PROGRAM MAIN
VAR
	Timer1 :TON;
	Timer2 : TON;
	Timer3 : TON;
	PulseTimer1 : TP;

	CurrentState  : States;
	
	ServoRTrigY : R_Trig ; 
	ServoRTrigX : R_Trig ; 
	
	//Eigen trigger booleans
	InitYReady : BOOL;
	InitXReady : BOOL;
	droppingDown : BOOL; //test
	
	TimerTest1 : TIME;
	TimerResult : TIME;
	
	Move_Arm : MoveArm;
	Count_Free_Spaces : CountFreeSpaces;
	Find_Free : FindFree;
	
	PalletArray: ARRAY [1..25] OF BOOL := [25(FALSE)];
	Pos : INT;
	
	DrinkArray: ARRAY [1..25] OF Drinks := [25(Drinks.Cola)]; 
	FreeCola : INT;
	FreeFanta : INT;
	
	//messages voor Nicky & Jens
	BottleAvailable : BOOL;
	NoCover : BOOL;
	NoBottle : BOOL;
	ColaFanta: INT;
	

	
END_VAR

PulseTimer1(IN:=GVL_IO.Start_button, PT:=T#150MS);
Timer1(IN:= GVL_IO.a_1_Vertical_Zaxis_downward, PT:= T#10MS);
Timer2(IN:=GVL_IO.a_1_Vertical_Zaxis_downward, PT:=T#10MS);
Timer3(IN:=droppingDown AND NOT GVL_IO.a_1_Vertical_Zaxis_downward, PT:=T#280MS);

CASE CurrentState OF
States.Init:
		//Aanzetten van servo's. Dit kan even duren GEEN HOMING
		GVL_IO.SVONX_SERVO_ON_tableX 	  := TRUE; 
		GVL_IO.SVONY_SERVO_ON_translY 	  := TRUE;
		
		GVL_IO.SETUPX_ORIGIN_tableX := PulseTimer1.Q;
		GVL_IO.SETUPY_ORIGIN_translY := PulseTimer1.Q;
		
		//// Koppelen van outputs Busy aan var's. Triggered op een falling edge.
		IF PulseTimer1.Q THEN
			ServoRTrigX ( clk := gvl_io.SETONX_ORIGIN_tableX ); 
	  		ServoRTrigY ( clk := gvl_io.SETONY_ORIGIN_translationY );
		END_IF
		
		// Bools setten aan de hand van triggers.
		IF ServoRTrigX.Q THEN
			InitXReady:= TRUE;
		END_IF
		
		IF ServoRTrigY.Q THEN
			InitYReady:= TRUE;
		END_IF
		
		// Init voltooid ga naar idle
		IF InitXReady AND InitYReady THEN
			Pos:= 1;
			NoCover := FALSE;
			NoBottle := FALSE;
			ColaFanta := drinks.Cola;
			CurrentState:= States.Idle;
		END_IF
		
States.Idle:
		//TEST =========================================================
		IF NOT GVL_IO.Stop_button THEN
			BottleAvailable := TRUE;
		END_IF
		//==============================================================
		Count_Free_Spaces(DrinkArray:=DrinkArray, PalletArray:= PalletArray);
		FreeCola := Count_Free_Spaces.FreeCola;
		FreeFanta := Count_Free_Spaces.FreeFanta;
		IF BottleAvailable AND GVL_IO.dp1_Can_detection AND GVL_IO.dp2_Cover_detection THEN
			Find_Free(DrinkArray:=DrinkArray, PalletArray:= PalletArray, TempDrink:= ColaFanta);
			Pos := Find_Free.FreePosition;
			NoCover := FALSE;
			NoBottle := FALSE;
			BottleAvailable := FALSE;
			CurrentState := States.MoveToPickUp;
		ELSIF BottleAvailable AND NOT GVL_IO.dp2_Cover_detection THEN
			NoCover := TRUE;
			BottleAvailable := FALSE;
		ELSIF BottleAvailable AND NOT GVL_IO.dp1_Can_detection THEN
			NoBottle := TRUE;
			BottleAvailable := FALSE;
		END_IF
		
States.MoveToPickUp:
		Move_Arm(Position:= 30);
		IF Move_Arm.OnNewLocation THEN
			CurrentState := States.PickUpDown;
		END_IF
		
States.PickUpDown:
		IF GVL_IO.a_0_Vertical_Zaxis_upward THEN
			GVL_IO.Aplus_Vert_axis_downwards := TRUE;
		END_IF
		
		IF GVL_IO.a_1_Vertical_Zaxis_downward THEN
			GVL_IO.Vplus_Vacuum_start := TRUE;
			
			IF Timer1.Q THEN
			CurrentState := States.PickUpUp;
			END_IF
		END_IF

States.PickUpUp:
		GVL_IO.Aplus_Vert_axis_downwards := FALSE;
		
		IF GVL_IO.a_0_Vertical_Zaxis_upward THEN
			CurrentState := States.Moving;
		END_IF
		
States.Moving:
		IF GVL_IO.a_0_Vertical_Zaxis_upward THEN
		
		Move_Arm(Position:= Pos);
		IF Move_Arm.OnNewLocation THEN
			PalletArray[Pos] := TRUE; // TEMP Cihan
			CurrentState := States.DropDown;
		END_IF
		END_IF
		
States.DropDown:
		IF GVL_IO.a_0_Vertical_Zaxis_upward THEN
			GVL_IO.Aplus_Vert_axis_downwards := TRUE;
			droppingDown := TRUE;
			TimerTest1 := TIME();
		END_IF
		
		
		IF 	GVL_IO.a_1_Vertical_Zaxis_downward THEN
			GVL_IO.Vplus_Vacuum_start := FALSE;
			IF Timer2.Q THEN
				TimerResult := TIME() - TimerTest1;
				droppingDown := FALSE;
				CurrentState := States.DropUp;
			END_IF
			
		ELSE IF Timer3.Q  THEN
		GVL_io.Aplus_Vert_axis_downwards := FALSE;
		droppingDown := FALSE;
		CurrentState := States.ManualCheck;
		END_IF
		END_IF

States.DropUp:
		IF GVL_IO.a_1_Vertical_Zaxis_downward THEN
			GVL_IO.Aplus_Vert_axis_downwards := FALSE;
		END_IF
		
		IF GVL_IO.a_0_Vertical_Zaxis_upward THEN
			CurrentState := States.Idle;
		END_IF
		
States.ManualCheck:
		GVL_IO.BR_Alarm_light := TRUE;
		GVL_io.Vplus_Vacuum_start := FALSE;
		IF GVL_IO.Reset_button THEN
			GVL_IO.BR_Alarm_light := FALSE;
			Currentstate := States.Idle;
		END_IF
END_CASE

END_PROGRAM

(* stored: Version 1.1.0.1, ProductVersion 3.1.4022.12
   POU MAIN: Id {a4f99ad4-3d99-4cc3-aec6-4b8f25d45e95}, SpecialFunc None *)
